(* Logix 5000 project; controller Commerford_topping_5477_V3 vendor 1 type 14 code 222 rev 33.11; software revision 33.02; part 6 of 6 *)
(* tags used below, declared in another part *)
   Master_Recipe : MasterRecipeSelect;
   PackML : ISA_TR_88_00_02;
   Proces : ProcessHandler;
   ProcessStates : DINT[32];
   Recipe : RecipeManager[4];
(* UN6_Object, continued *)

ROUTINE Process_Management   (* ladder *)
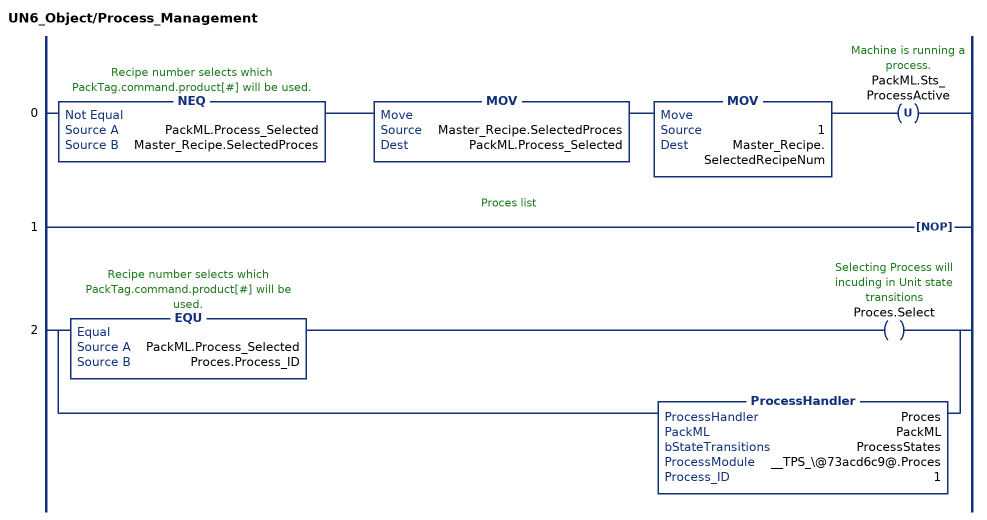
   0: NEQ(PackML.Process_Selected,Master_Recipe.SelectedProces)MOV(Master_Recipe.SelectedProces,PackML.Process_Selected)MOV(1,Master_Recipe.SelectedRecipeNum)OTU(PackML.Sts_ProcessActive);
   // Proces list
   1: NOP();
   2: [EQU(PackML.Process_Selected,Proces.Process_ID) OTE(Proces.Select) ,ProcessHandler(Proces,PackML,ProcessStates,__TPS_\@73acd6c9@.Proces,1) ];
END_ROUTINE

ROUTINE Recipe_Management   (* ladder *)
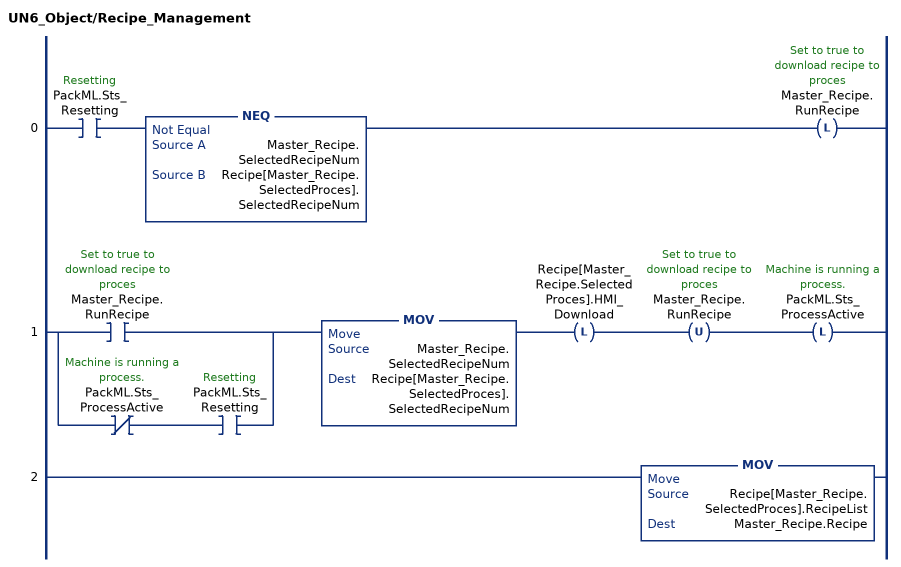
   0: XIC(PackML.Sts_Resetting)NEQ(Master_Recipe.SelectedRecipeNum,Recipe[Master_Recipe.SelectedProces].SelectedRecipeNum)OTL(Master_Recipe.RunRecipe);
   1: [XIC(Master_Recipe.RunRecipe) ,XIO(PackML.Sts_ProcessActive) XIC(PackML.Sts_Resetting) ]MOV(Master_Recipe.SelectedRecipeNum,Recipe[Master_Recipe.SelectedProces].SelectedRecipeNum)OTL(Recipe[Master_Recipe.SelectedProces].HMI_Download)OTU(Master_Recipe.RunRecipe)OTL(PackML.Sts_ProcessActive);
   2: MOV(Recipe[Master_Recipe.SelectedProces].RecipeList,Master_Recipe.Recipe);
END_ROUTINE
END_PROGRAM
